PROGRAM MAIN
VAR
END_VAR

END_PROGRAM

(* stored: Version 1.1.0.1
   POU MAIN: Id {c31c8014-acb9-42a7-9d85-2715814808ce} *)
